// TwinCAT 3 PLC project M1K4_PLC
// ProgramVersion: 3.1.4020.5
// libraries:
//   Tc2_MC2, * (Beckhoff Automation GmbH)
//   Tc2_Standard, * (Beckhoff Automation GmbH)
//   Tc2_System, * (Beckhoff Automation GmbH)
//   Tc2_Utilities, * (Beckhoff Automation GmbH)
//   Tc3_Module, * (Beckhoff Automation GmbH)
//   VisuDialogs
//   lcls-twincat-motion,0.0.0,SLAC
// project tree:
//   DUTs/ DUT_MotionStage_Extras.TcDUT (not stored)
//   / GlobalTextList.TcGTLO, PlcTask.TcTTO, Visualization Manager.TcVMO (not stored)
//   POUs/ MAIN.TcPOU
//   VISUs/ Visualization.TcVIS, VISU_MotionStage.TcVIS (not stored)
// real-time tasks:
//   TASK PlcTask: cycle T#10ms, priority 20, ADS port 350
// motion (NC):
// I/O:
//   DEVICE Device 3 (EtherCAT), AmsNetId 172.21.148.46.4.1
//     Term 1 (EK1100) [EK1100 EtherCAT Coupler (2A E-Bus)]
//       Term 2 (EL7041-1000) - Xup
//       Term 3 (EL7041-1000) - Xdwn
//       Term 4 (EL7041-1000) - Yup [EL7041-1000 1Ch. Stepper motor output stage (50V, 5A, standard)]
//       Term 5 (EL7041-1000) - Ydwn [EL7041-1000 1Ch. Stepper motor output stage (50V, 5A, standard)]
//       Term 6 (EL7041-1000) - PitchCoarse
//       Term 7 (EL7041-1000) - Bender
//       Term 8 (EL6001) - PitchFine [EL6001 Interface (RS232)]
//       Term 9 (EL5042) - X
//       Term 10 (EL5042) - Y
//       Term 11 (EL5042) - PitchBender
//       Term 12 (EL1004) - STO
//       Term 13 (EL9505) - BenderLim
//       Term 14 (EL9011)
// variable links:
//   M1K4_PLC Instance <-> Device 3 (EtherCAT)/Term 1 (EK1100)/Term 10 (EL5042) - Y
//     PlcTask Inputs/MAIN.y_dwn_enc/Count <-> FB Inputs Channel 2/Position
//     PlcTask Inputs/MAIN.y_up_enc/Count <-> FB Inputs Channel 1/Position
//   M1K4_PLC Instance <-> Device 3 (EtherCAT)/Term 1 (EK1100)/Term 12 (EL1004) - STO
//     PlcTask Inputs/MAIN.bSTOEnable1 <-> Channel 1/Input
//     PlcTask Inputs/MAIN.bSTOEnable2 <-> Channel 2/Input
//   M1K4_PLC Instance <-> Device 3 (EtherCAT)/Term 1 (EK1100)/Term 2 (EL7041-1000) - Xup
//     PlcTask Inputs/MAIN.M3.bLimitBackwardEnable <-> STM Status/Status/Digital input 2
//     PlcTask Inputs/MAIN.M3.bLimitForwardEnable <-> STM Status/Status/Digital input 1
//   M1K4_PLC Instance <-> Device 3 (EtherCAT)/Term 1 (EK1100)/Term 3 (EL7041-1000) - Xdwn
//     PlcTask Inputs/MAIN.M4.bLimitBackwardEnable <-> STM Status/Status/Digital input 2
//     PlcTask Inputs/MAIN.M4.bLimitForwardEnable <-> STM Status/Status/Digital input 1
//   M1K4_PLC Instance <-> Device 3 (EtherCAT)/Term 1 (EK1100)/Term 4 (EL7041-1000) - Yup
//     PlcTask Inputs/MAIN.M1.bLimitBackwardEnable <-> STM Status/Status/Digital input 2
//     PlcTask Inputs/MAIN.M1.bLimitForwardEnable <-> STM Status/Status/Digital input 1
//   M1K4_PLC Instance <-> Device 3 (EtherCAT)/Term 1 (EK1100)/Term 5 (EL7041-1000) - Ydwn
//     PlcTask Inputs/MAIN.M2.bLimitBackwardEnable <-> STM Status/Status/Digital input 2
//     PlcTask Inputs/MAIN.M2.bLimitForwardEnable <-> STM Status/Status/Digital input 1
//   M1K4_PLC Instance <-> Device 3 (EtherCAT)/Term 1 (EK1100)/Term 6 (EL7041-1000) - PitchCoarse
//     PlcTask Inputs/MAIN.M5.bLimitBackwardEnable <-> STM Status/Status/Digital input 2
//     PlcTask Inputs/MAIN.M5.bLimitForwardEnable <-> STM Status/Status/Digital input 1
//   M1K4_PLC Instance <-> Device 3 (EtherCAT)/Term 1 (EK1100)/Term 7 (EL7041-1000) - Bender
//     PlcTask Inputs/MAIN.M6.bLimitBackwardEnable <-> STM Status/Status/Digital input 2
//     PlcTask Inputs/MAIN.M6.bLimitForwardEnable <-> STM Status/Status/Digital input 1
//   M1K4_PLC Instance <-> Device 3 (EtherCAT)/Term 1 (EK1100)/Term 9 (EL5042) - X
//     PlcTask Inputs/MAIN.x_dwn_enc/Count <-> FB Inputs Channel 2/Position
//     PlcTask Inputs/MAIN.x_up_enc/Count <-> FB Inputs Channel 1/Position
//   M1K4_PLC Instance <-> NC-Task 1 SAF/Axes/Axis_Bender
//     PlcTask Inputs/MAIN.M6.Axis.NcToPlc <-> Outputs/ToPlc
//     PlcTask Outputs/MAIN.M6.Axis.PlcToNc <-> Inputs/FromPlc
//   M1K4_PLC Instance <-> NC-Task 1 SAF/Axes/Axis_PitchCoarse
//     PlcTask Inputs/MAIN.M5.Axis.NcToPlc <-> Outputs/ToPlc
//     PlcTask Outputs/MAIN.M5.Axis.PlcToNc <-> Inputs/FromPlc
//   M1K4_PLC Instance <-> NC-Task 1 SAF/Axes/Axis_Xdwn
//     PlcTask Inputs/MAIN.M4.Axis.NcToPlc <-> Outputs/ToPlc
//     PlcTask Outputs/MAIN.M4.Axis.PlcToNc <-> Inputs/FromPlc
//   M1K4_PLC Instance <-> NC-Task 1 SAF/Axes/Axis_Xup
//     PlcTask Inputs/MAIN.M3.Axis.NcToPlc <-> Outputs/ToPlc
//     PlcTask Outputs/MAIN.M3.Axis.PlcToNc <-> Inputs/FromPlc
//   M1K4_PLC Instance <-> NC-Task 1 SAF/Axes/Axis_Ydwn
//     PlcTask Inputs/MAIN.M2.Axis.NcToPlc <-> Outputs/ToPlc
//     PlcTask Outputs/MAIN.M2.Axis.PlcToNc <-> Inputs/FromPlc
//   M1K4_PLC Instance <-> NC-Task 1 SAF/Axes/Axis_Yup
//     PlcTask Inputs/MAIN.M1.Axis.NcToPlc <-> Outputs/ToPlc
//     PlcTask Outputs/MAIN.M1.Axis.PlcToNc <-> Inputs/FromPlc

CONFIGURATION M1K4_PLC
    RESOURCE PLC ON TwinCAT3
        TASK PlcTask(INTERVAL := T#10ms, PRIORITY := 20);
        PROGRAM MAIN WITH PlcTask : MAIN;
    END_RESOURCE
END_CONFIGURATION

// ---- POUs/MAIN.TcPOU
PROGRAM MAIN
VAR		
    M1: DUT_MotionStage:=(nCommand:=3); // Yup
	M2: DUT_MotionStage:=(nCommand:=3); // Ydwn
	M3: DUT_MotionStage:=(nCommand:=3); // Xup
	M4: DUT_MotionStage:=(nCommand:=3); // Xdwn
	M5: DUT_MotionStage:=(nCommand:=3); // PitchCoarse
	M6: DUT_MotionStage:=(nCommand:=3); // Bender

	// Axis_Extras Structs
	M1_Extras : DUT_MotionStage_Extras;
	M2_Extras : DUT_MotionStage_Extras;
	M3_Extras : DUT_MotionStage_Extras;
	M4_Extras : DUT_MotionStage_Extras;
	M5_Extras : DUT_MotionStage_Extras;

	fbMotionStage_x_up, fbMotionStage_x_dwn, fbMotionStage_y_up, fbMotionStage_y_dwn, fbMotionStage_pitch, fbMotionStage_bender : FB_MotionStage;

	bSTOEnable1 AT %I* : BOOL;
	bSTOEnable2 AT %I* : BOOL;

	x_up_enc  AT %I*: ST_RenishawAbsEnc;
	x_dwn_enc  AT %I*: ST_RenishawAbsEnc;

	y_up_enc  AT %I*: ST_RenishawAbsEnc;
	y_dwn_enc  AT %I*: ST_RenishawAbsEnc;

	// Auto coupling function block
	fbAutoCoupleX : FB_GantryAutoCoupling;
	fbAutoCoupleY : FB_GantryAutoCoupling;

	bExecuteCoupleX : BOOL;
	bExecuteCoupleY : BOOL;
	bExecuteDecoupleX : BOOL;
	bExecuteDecoupleY : BOOL;
	bGantryAlreadyCoupledX : BOOL;
	bGantryAlreadyCoupledY : BOOL;
	
	// Gantry variables
	nCurrGantryX : LINT;
	nCurrGantryY : LINT;
	nGantryTolX : LINT := 50000;
	nGantryTolY : LINT := 50000;
END_VAR

// M1K4
// Buttons to enable motors: write 0 to enable, 2 to disable
M1.nEnableMode; // Yup
M2.nEnableMode; // Ydwn
M3.nEnableMode; // Xup
M4.nEnableMode; // Xdwn
M5.nEnableMode; // PitchCoarse

// Encoder Reference Values: Starting motor positions prior to checkout
(*
y_up_enc.Ref := 4411200;
y_dwn_enc.Ref := 4084980;
*)
// Post-alignment reference values
y_up_enc.Ref := 15000270;
y_dwn_enc.Ref := 15454300;
x_up_enc.Ref := 24000300;
x_dwn_enc.Ref := 23999400;

// Gantry Differences to monitor
nCurrGantryY := ((ULINT_TO_LINT(y_up_enc.Count) - ULINT_TO_LINT(y_up_enc.Ref)) - (ULINT_TO_LINT(y_dwn_enc.Count) - ULINT_TO_LINT(y_dwn_enc.Ref)));
nCurrGantryX := ((ULINT_TO_LINT(x_up_enc.Count) - ULINT_TO_LINT(x_up_enc.Ref)) - (ULINT_TO_LINT(x_dwn_enc.Count) - ULINT_TO_LINT(x_dwn_enc.Ref)));

// E-stop
M1.bHardwareEnable := bSTOEnable1 AND bSTOEnable2;
M2.bHardwareEnable := bSTOEnable1 AND bSTOEnable2;
M3.bHardwareEnable := bSTOEnable1 AND bSTOEnable2;
M4.bHardwareEnable := bSTOEnable1 AND bSTOEnable2;
M5.bHardwareEnable := bSTOEnable1 AND bSTOEnable2;
M6.bHardwareEnable := bSTOEnable1 AND bSTOEnable2;

// Start Autocoupling
fbAutoCoupleX(nGantryTol:=nGantryTolX, Master:=M3, MasterEnc:=x_up_enc, Slave:=M4,
	          SlaveEnc:=x_dwn_enc, bExecuteCouple:=bExecuteCoupleX,
              bExecuteDecouple:=bExecuteDecoupleX,
              bGantryAlreadyCoupled=>bGantryAlreadyCoupledX);

fbAutoCoupleY(nGantryTol:=nGantryTolY, Master:=M1, MasterEnc:=y_up_enc, Slave:=M2,
	          SlaveEnc:=y_dwn_enc, bExecuteCouple:=bExecuteCoupleY,
              bExecuteDecouple:=bExecuteDecoupleY,
			  bGantryAlreadyCoupled=>bGantryAlreadyCoupledY);

fbMotionStage_y_up  (stMotionStage:=M1);
fbMotionStage_y_dwn (stMotionStage:=M2);
fbMotionStage_x_up  (stMotionStage:=M3);
fbMotionStage_x_dwn (stMotionStage:=M4);
fbMotionStage_pitch (stMotionStage:=M5);
fbMotionStage_bender (stMotionStage:=M6);

END_PROGRAM

// ---- GlobalTextList.TcGTLO
TEXTLIST GlobalTextList
  366 = '%f'
  20 = '%X'
  12 = '+'
  6 = '-'
  16 = '0 = Default Acceleration'
  18 = '0 = Default Deceleration'
  15 = 'Acceleration: %f'
  317 = 'Already Coupled: %f'
  10 = 'Clear'
  370 = 'Control'
  323 = 'Couple Motors'
  658 = 'Couple Status: 0 = Decoupled, 1 = Coupled'
  318 = 'Couple Status: TRUE if coupled'
  660 = 'Current Gantry Difference (Axilon): %f'
  128 = 'Current Gantry Difference in nm'
  320 = 'Current Gantry Difference in um'
  319 = 'Current Gantry Difference: %f'
  367 = 'Current Position'
  17 = 'Deceleration: %f'
  321 = 'Decouple Motors'
  24 = 'Disable'
  25 = 'Enable'
  22 = 'Enable Mode: %f'
  657 = 'Enable Status: 0 = Enabled, 2 = Disabled'
  659 = 'Ensure motors are coupled before attempting motion!'
  21 = 'Error Code'
  19 = 'Error:'
  8 = 'GO'
  9 = 'GO to set position'
  368 = 'High Limit Hit Indicator'
  365 = 'Low Limit Hit Indicator'
  329 = 'mm'
  369 = 'Moving:'
  479 = 'Pitch - MASTER'
  324 = 'Press To Couple Motors'
  322 = 'Press To Decouple Motors for independent control'
  5 = 'Set Position'
  13 = 'Settings'
  364 = 'Status'
  7 = 'Step Size'
  11 = 'STOP'
  380 = 'Units: mm'
  825 = 'Units: mmUnits: um'
  480 = 'Units: um'
  558 = 'Units: Units: mm'
  481 = 'Units: urad'
  14 = 'Velocity: %f'
  23 = 'Write 0 to Enable, 2 to Disable'
  326 = 'Xdwn - SLAVE'
  325 = 'Xup - MASTER'
  880 = 'Ydwn - SLAVE'
  315 = 'Yleft - MASTER'
  316 = 'Yright - SLAVE'
  993 = 'Yup - MASTER'
END_TEXTLIST

// ---- VISUs/Visualization.TcVIS
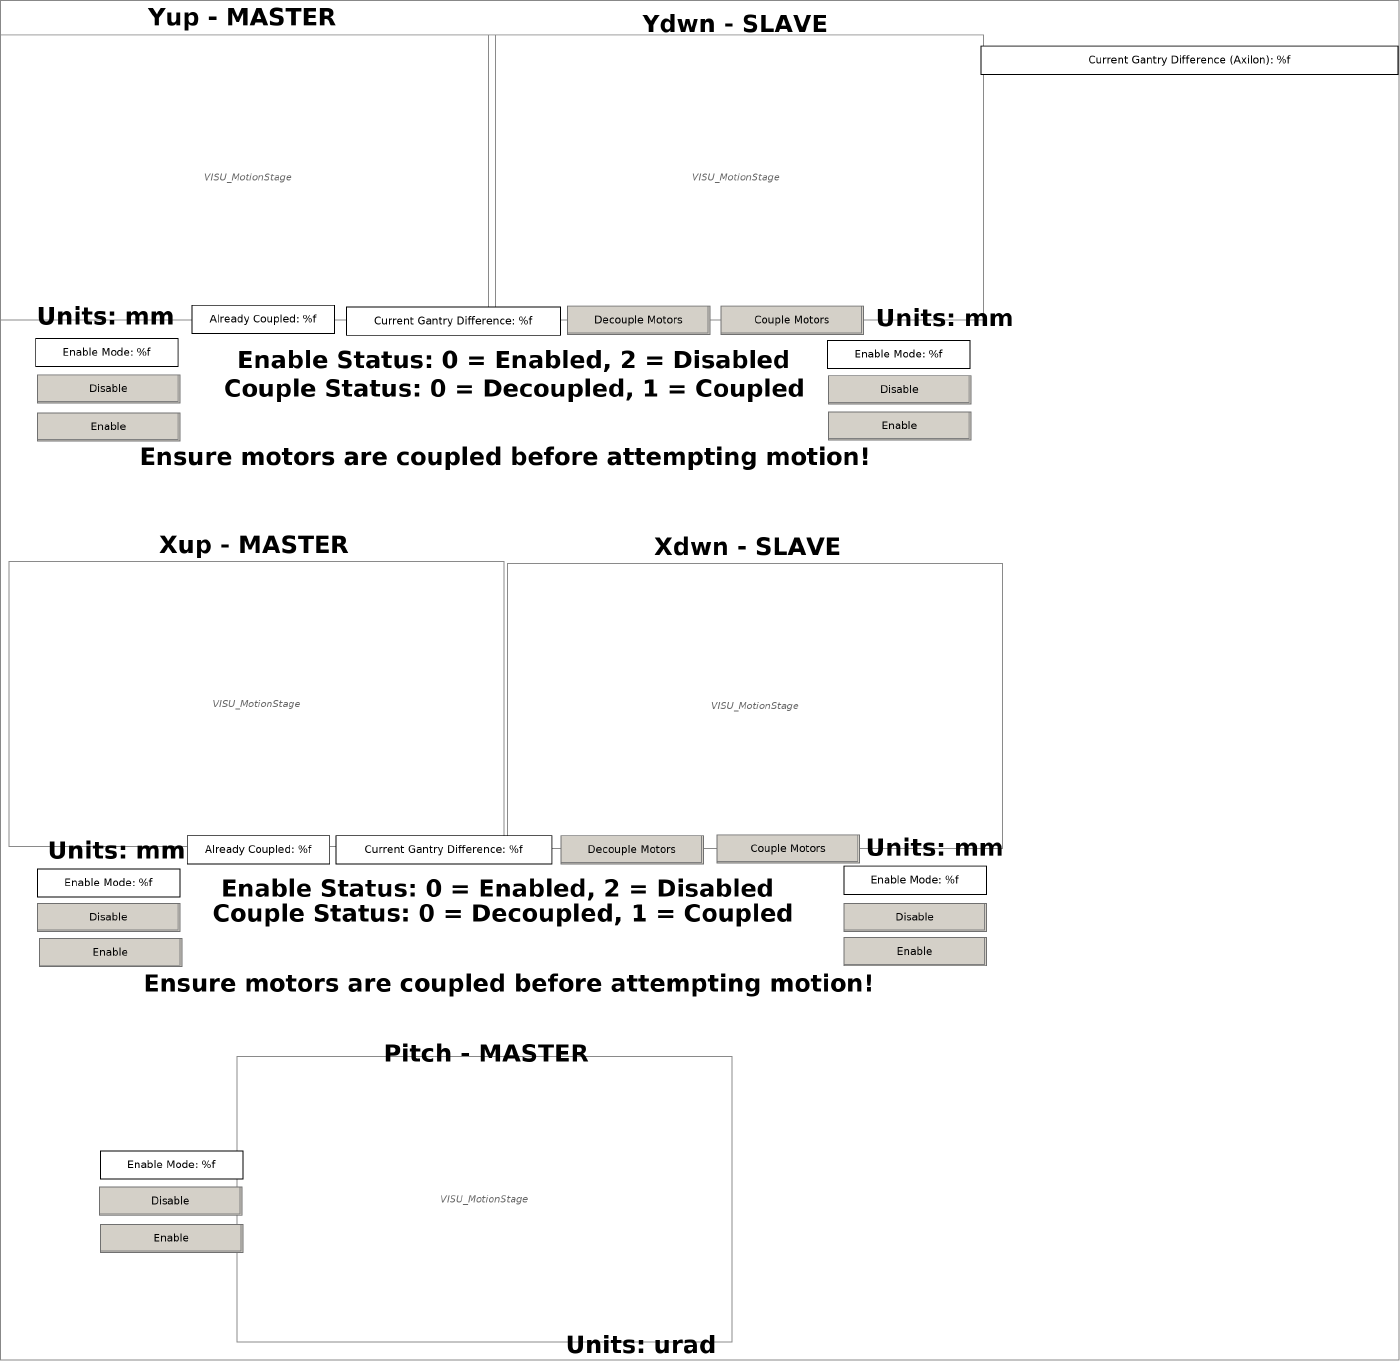
VISUALIZATION Visualization  // 1469x1429
    Label (14,2 481x31), "Yup - MASTER"
    Frame (0,36 520x300)
        shows VISU_MotionStage(VisuMotionStage := MAIN.M1, Extras := MAIN.M1_Extras)
    Frame (512,36 520x300)
        shows VISU_MotionStage(VisuMotionStage := MAIN.M2, Extras := MAIN.M2_Extras)
    Label (531,9 481x31), "Ydwn - SLAVE"
    Rectangle (201,320 150x30), "Already Coupled: %f", tooltip "Couple Status: TRUE if coupled", text variable: MAIN.bGantryAlreadyCoupledY
    Rectangle (363,322 225x30), "Current Gantry Difference: %f", tooltip "Current Gantry Difference in nm", text variable: MAIN.nCurrGantryY
    Button (756,321 150x30), "Couple Motors", tooltip "Press To Couple Motors", text variable: MAIN.bExecuteCoupleY
        OnMouseDown: execute { MAIN.bExecuteCoupleY := TRUE; }
    Frame (9,589 520x300)
        shows VISU_MotionStage(VisuMotionStage := MAIN.M3, Extras := MAIN.M3_Extras)
    Label (26,556 481x31), "Xup - MASTER"
    Frame (532,591 520x300)
        shows VISU_MotionStage(VisuMotionStage := MAIN.M4, Extras := MAIN.M4_Extras)
    Label (544,558 481x31), "Xdwn - SLAVE"
    Rectangle (196,877 150x30), "Already Coupled: %f", tooltip "Couple Status: TRUE if coupled", text variable: MAIN.bGantryAlreadyCoupledX
    Rectangle (352,877 227x30), "Current Gantry Difference: %f", tooltip "Current Gantry Difference in nm", text variable: MAIN.nCurrGantryX
    Frame (248,1109 520x300)
        shows VISU_MotionStage(VisuMotionStage := MAIN.M5, Extras := MAIN.M5_Extras)
    Label (270,1090 481x31), "Pitch - MASTER"
    Label (31,316 160x31), "Units: mm"
    Label (916,318 151x31), "Units: mm"
    Label (27,877 191x31), "Units: mm"
    Label (894,874 174x31), "Units: mm"
    Label (595,1396 155x31), "Units: urad"
    Rectangle (37,355 150x30), "Enable Mode: %f", tooltip "Write 0 to Enable, 2 to Disable", text variable: MAIN.M1.nEnableMode
    Rectangle (868,357 150x30), "Enable Mode: %f", tooltip "Write 0 to Enable, 2 to Disable", text variable: MAIN.M2.nEnableMode
    Button (595,321 150x30), "Decouple Motors", tooltip "Press To Decouple Motors for independent control"
        OnMouseDown: execute { MAIN.bExecuteDecoupleY := TRUE; }
    Button (39,393 150x30), "Disable"
        OnMouseDown: execute { MAIN.M1.nEnableMode := 2; }
    Button (39,433 150x30), "Enable", colour toggle: MAIN.bExecuteDecoupleY
        OnMouseDown: execute { MAIN.M1.nEnableMode := 0; }
    Button (869,394 150x30), "Disable"
        OnMouseDown: execute { MAIN.M2.nEnableMode := 2; }
    Button (869,432 150x30), "Enable", colour toggle: MAIN.bExecuteDecoupleY
        OnMouseDown: execute { MAIN.M2.nEnableMode := 0; }
    Button (588,877 150x30), "Decouple Motors", tooltip "Press To Decouple Motors for independent control"
        OnMouseDown: execute { MAIN.bExecuteDecoupleX := TRUE; }
    Button (752,876 150x30), "Couple Motors", tooltip "Press To Couple Motors", text variable: MAIN.bExecuteCoupleY
        OnMouseDown: execute { MAIN.bExecuteCoupleX := TRUE; }
    Rectangle (39,912 150x30), "Enable Mode: %f", tooltip "Write 0 to Enable, 2 to Disable", text variable: MAIN.M3.nEnableMode
    Button (39,948 150x30), "Disable"
        OnMouseDown: execute { MAIN.M3.nEnableMode := 2; }
    Button (41,985 150x30), "Enable", colour toggle: MAIN.bExecuteDecoupleY
        OnMouseDown: execute { MAIN.M3.nEnableMode := 0; }
    Rectangle (885,909 150x30), "Enable Mode: %f", tooltip "Write 0 to Enable, 2 to Disable", text variable: MAIN.M4.nEnableMode
    Button (885,948 150x30), "Disable"
        OnMouseDown: execute { MAIN.M4.nEnableMode := 2; }
    Button (885,984 150x30), "Enable", colour toggle: MAIN.bExecuteDecoupleY
        OnMouseDown: execute { MAIN.M4.nEnableMode := 0; }
    Rectangle (105,1208 150x30), "Enable Mode: %f", tooltip "Write 0 to Enable, 2 to Disable", text variable: MAIN.M5.nEnableMode
    Button (104,1246 150x30), "Disable"
        OnMouseDown: execute { MAIN.M5.nEnableMode := 2; }
    Button (105,1285 150x30), "Enable", colour toggle: MAIN.bExecuteDecoupleY
        OnMouseDown: execute { MAIN.M5.nEnableMode := 0; }
    Label (255,362 568x31), "Enable Status: 0 = Enabled, 2 = Disabled"
    Label (247,392 586x31), "Couple Status: 0 = Decoupled, 1 = Coupled"
    Label (238,917 568x31), "Enable Status: 0 = Enabled, 2 = Disabled"
    Label (235,943 586x31), "Couple Status: 0 = Decoupled, 1 = Coupled"
    Label (150,464 760x30), "Ensure motors are coupled before attempting motion!"
    Label (154,1017 760x30), "Ensure motors are coupled before attempting motion!"
    Rectangle (1029,48 438x30), "Current Gantry Difference (Axilon): %f", tooltip "Current Gantry Difference in um", text variable: MAIN.fCurrGantryY_Axilon_um
END_VISUALIZATION
